// SIMATIC S7-200 project (STEP 7-Micro/WIN), CPU 224 UN REL 02.02

ORGANIZATION_BLOCK MAIN:OB1
TITLE=PROGRAM COMMENTS
BEGIN
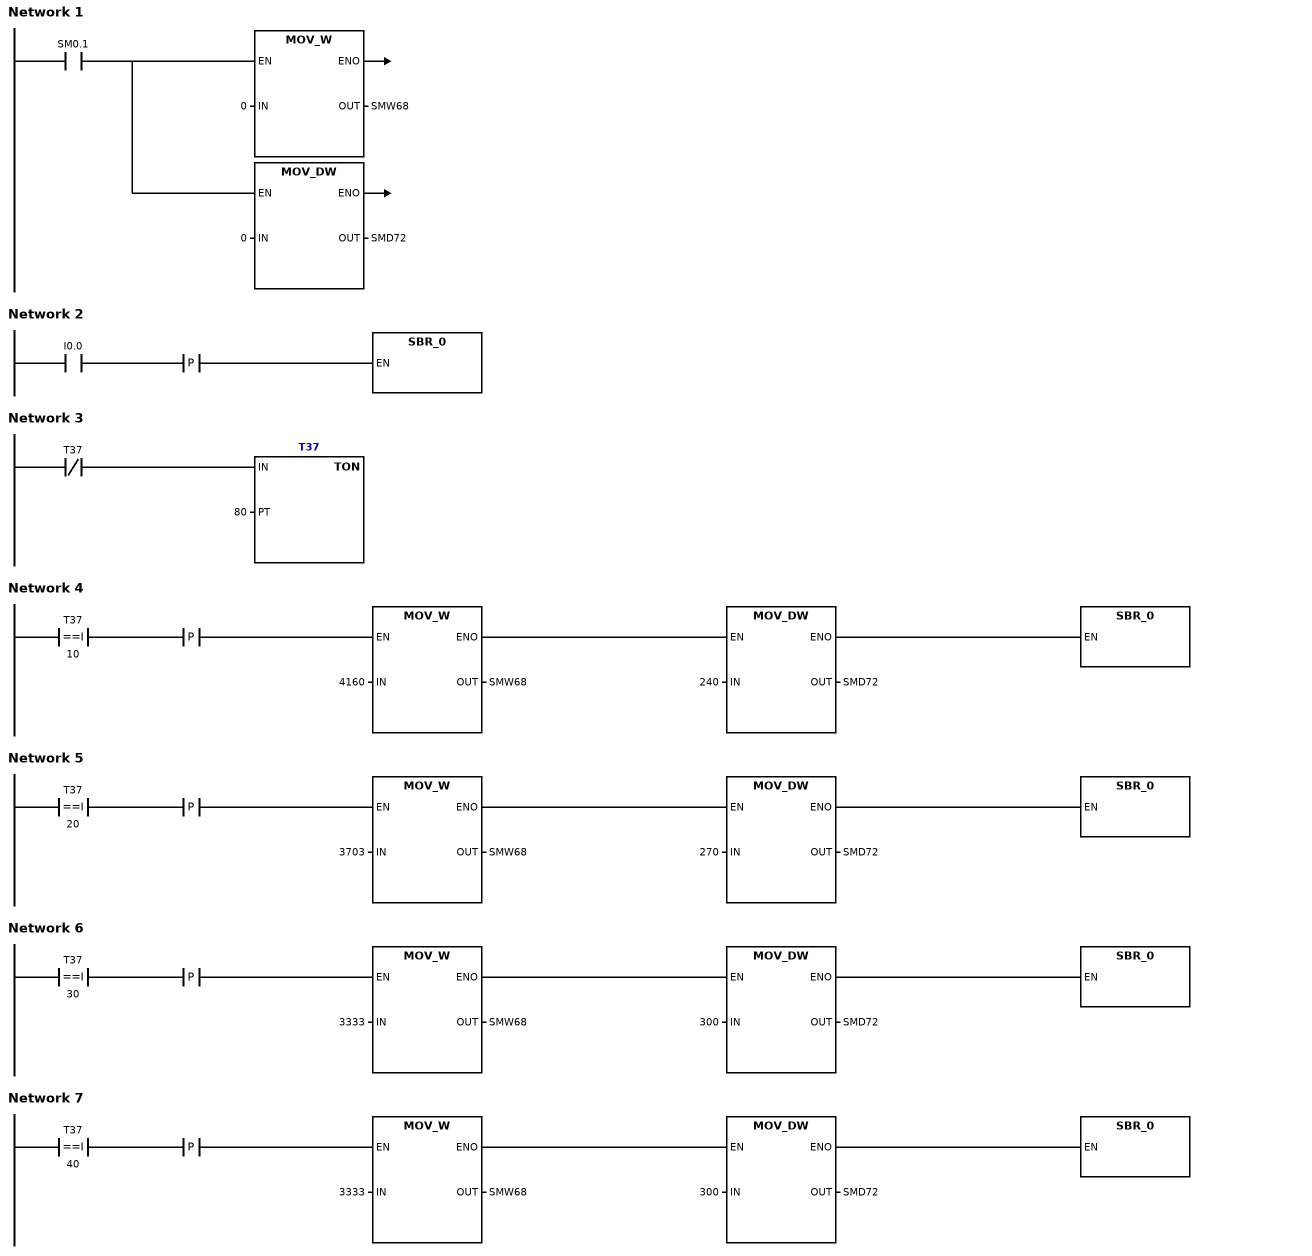
Network 1
LD     SM0.1
MOVW   0, SMW68
MOVD   0, SMD72
Network 2
LD     I0.0
EU
CALL   SBR_0:SBR0
Network 3
LDN    T37
TON    T37, 80
Network 4
LDW=   T37, 10
EU
MOVW   4160, SMW68
AENO
MOVD   240, SMD72
AENO
CALL   SBR_0:SBR0
Network 5
LDW=   T37, 20
EU
MOVW   3703, SMW68
AENO
MOVD   270, SMD72
AENO
CALL   SBR_0:SBR0
Network 6
LDW=   T37, 30
EU
MOVW   3333, SMW68
AENO
MOVD   300, SMD72
AENO
CALL   SBR_0:SBR0
Network 7
// (network saved uncompiled; LAD cells follow)
// row 0: c0 -|==I|- T37, 40  c1 -|P|-  c2 --  c3 [MOV_W EN:=power@row0, IN:=3333, ENO=>power, OUT=>SMW68]  c4 --  c5 --  c6 [MOV_DW EN:=power@row0, IN:=300, ENO=>power, OUT=>SMD72]  c7 --  c8 --  c9 [SBR_0 EN:=power@row0]
// row 1: c3 [box]  c6 [box]
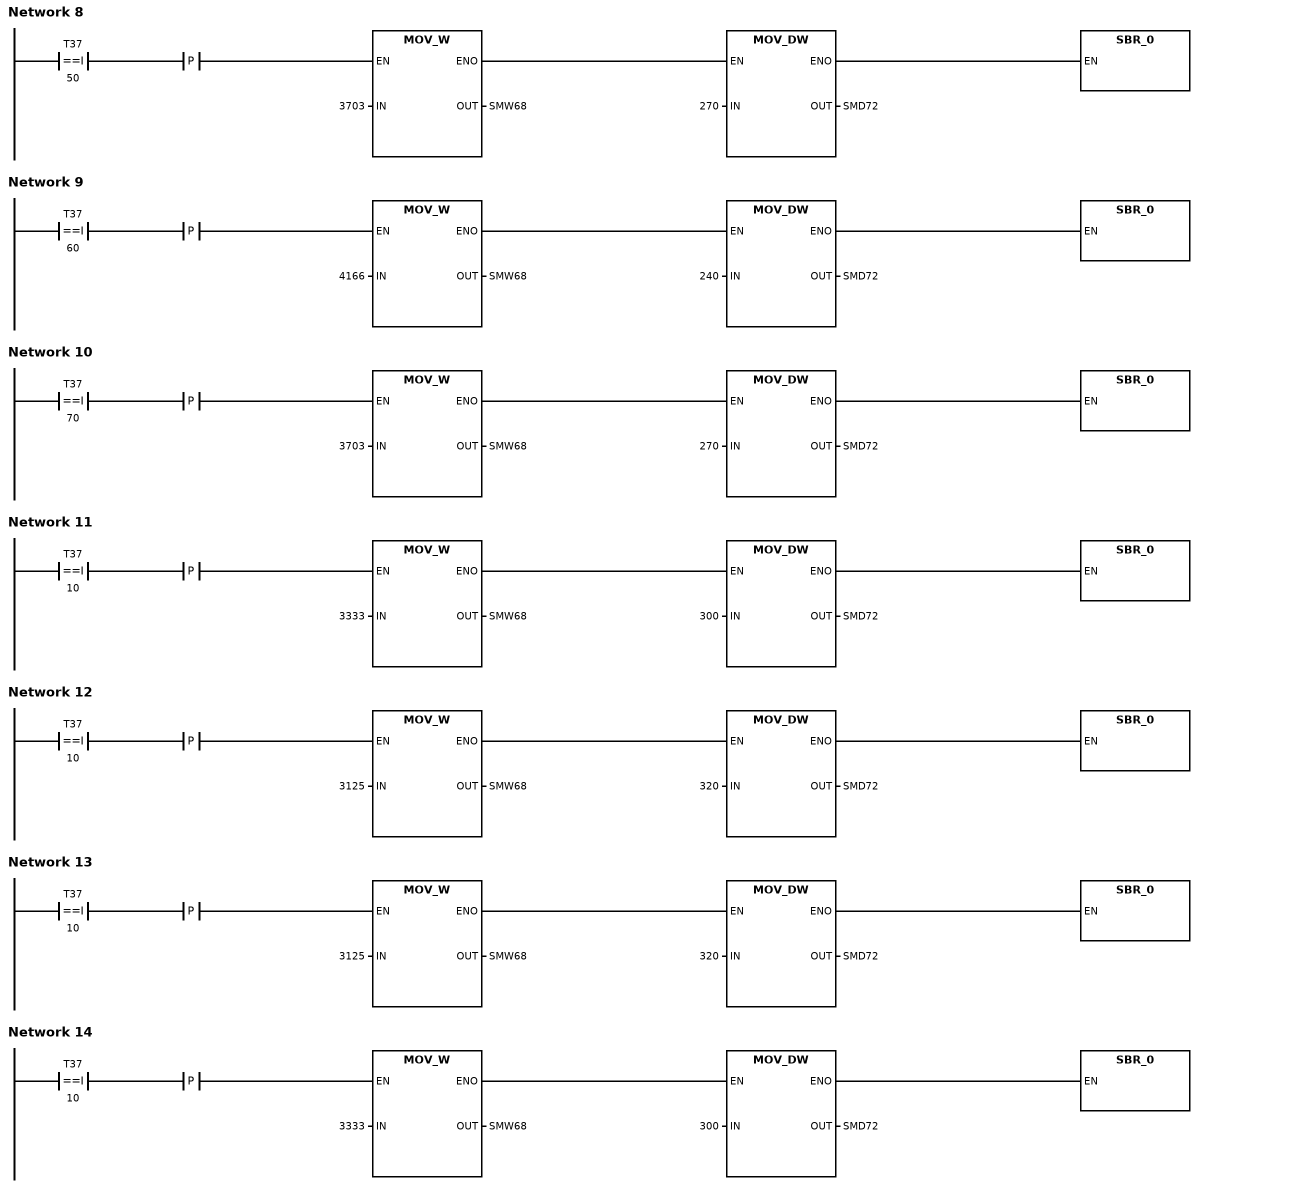
Network 8
// (network saved uncompiled; LAD cells follow)
// row 0: c0 -|==I|- T37, 50  c1 -|P|-  c2 --  c3 [MOV_W EN:=power@row0, IN:=3703, ENO=>power, OUT=>SMW68]  c4 --  c5 --  c6 [MOV_DW EN:=power@row0, IN:=270, ENO=>power, OUT=>SMD72]  c7 --  c8 --  c9 [SBR_0 EN:=power@row0]
// row 1: c3 [box]  c6 [box]
Network 9
// (network saved uncompiled; LAD cells follow)
// row 0: c0 -|==I|- T37, 60  c1 -|P|-  c2 --  c3 [MOV_W EN:=power@row0, IN:=4166, ENO=>power, OUT=>SMW68]  c4 --  c5 --  c6 [MOV_DW EN:=power@row0, IN:=240, ENO=>power, OUT=>SMD72]  c7 --  c8 --  c9 [SBR_0 EN:=power@row0]
// row 1: c3 [box]  c6 [box]
Network 10
// (network saved uncompiled; LAD cells follow)
// row 0: c0 -|==I|- T37, 70  c1 -|P|-  c2 --  c3 [MOV_W EN:=power@row0, IN:=3703, ENO=>power, OUT=>SMW68]  c4 --  c5 --  c6 [MOV_DW EN:=power@row0, IN:=270, ENO=>power, OUT=>SMD72]  c7 --  c8 --  c9 [SBR_0 EN:=power@row0]
// row 1: c3 [box]  c6 [box]
Network 11
LDW=   T37, 10
EU
MOVW   3333, SMW68
AENO
MOVD   300, SMD72
AENO
CALL   SBR_0:SBR0
Network 12
LDW=   T37, 10
EU
MOVW   3125, SMW68
AENO
MOVD   320, SMD72
AENO
CALL   SBR_0:SBR0
Network 13
LDW=   T37, 10
EU
MOVW   3125, SMW68
AENO
MOVD   320, SMD72
AENO
CALL   SBR_0:SBR0
Network 14
LDW=   T37, 10
EU
MOVW   3333, SMW68
AENO
MOVD   300, SMD72
AENO
CALL   SBR_0:SBR0
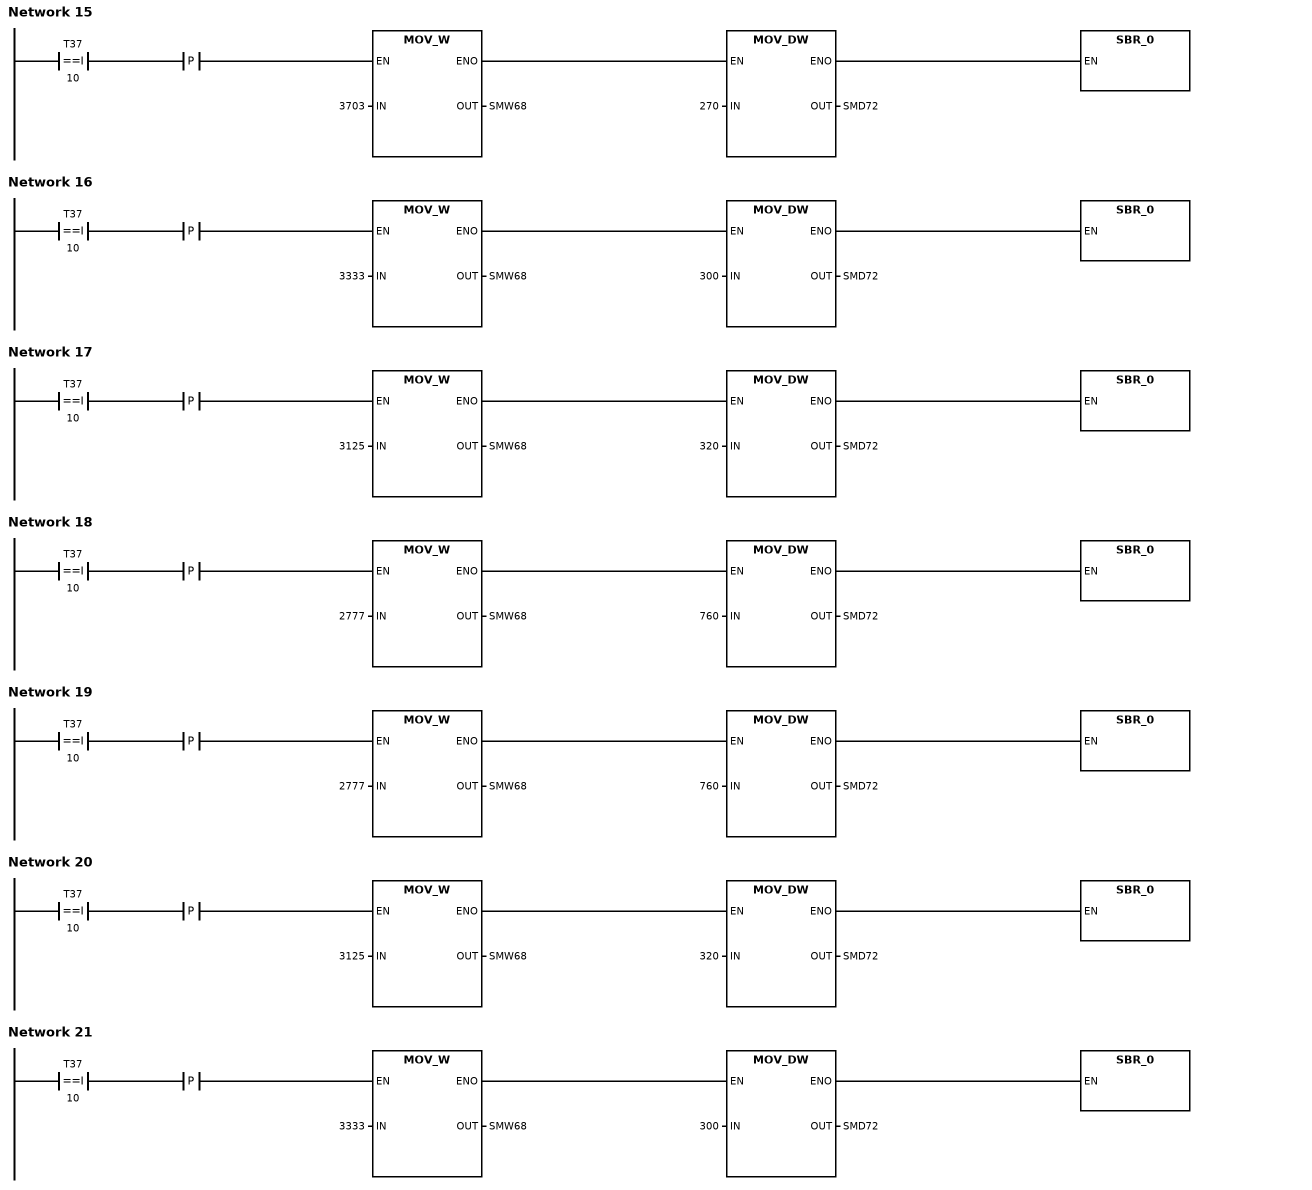
Network 15
LDW=   T37, 10
EU
MOVW   3703, SMW68
AENO
MOVD   270, SMD72
AENO
CALL   SBR_0:SBR0
Network 16
LDW=   T37, 10
EU
MOVW   3333, SMW68
AENO
MOVD   300, SMD72
AENO
CALL   SBR_0:SBR0
Network 17
LDW=   T37, 10
EU
MOVW   3125, SMW68
AENO
MOVD   320, SMD72
AENO
CALL   SBR_0:SBR0
Network 18
LDW=   T37, 10
EU
MOVW   2777, SMW68
AENO
MOVD   760, SMD72
AENO
CALL   SBR_0:SBR0
Network 19
LDW=   T37, 10
EU
MOVW   2777, SMW68
AENO
MOVD   760, SMD72
AENO
CALL   SBR_0:SBR0
Network 20
LDW=   T37, 10
EU
MOVW   3125, SMW68
AENO
MOVD   320, SMD72
AENO
CALL   SBR_0:SBR0
Network 21
LDW=   T37, 10
EU
MOVW   3333, SMW68
AENO
MOVD   300, SMD72
AENO
CALL   SBR_0:SBR0
END_ORGANIZATION_BLOCK

SUBROUTINE_BLOCK SBR_0:SBR0
TITLE=SUBROUTINE COMMENTS
BEGIN
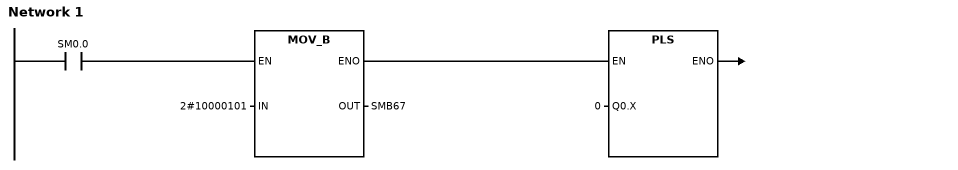
Network 1
LD     SM0.0
MOVB   2#10000101, SMB67
AENO
PLS    0
Network 2 // Network Title
// Network Comment
END_SUBROUTINE_BLOCK
